PROGRAM Auto
VAR
	MovRightS: BOOL;
	MovRightL: BOOL;
	MovLeftS: BOOL;
	TON_Right: TON;
	TON_Left: TON;
	
	Home: BOOL;
	HomeMemory: BOOL;
	ManRequest: BOOL;
	TON_Right1: TON;
	TON_Left1: TON;
END_VAR
VAR // added by the converter: edge detectors and wires of the graphical bodies
    _w1 : BOOL;
END_VAR

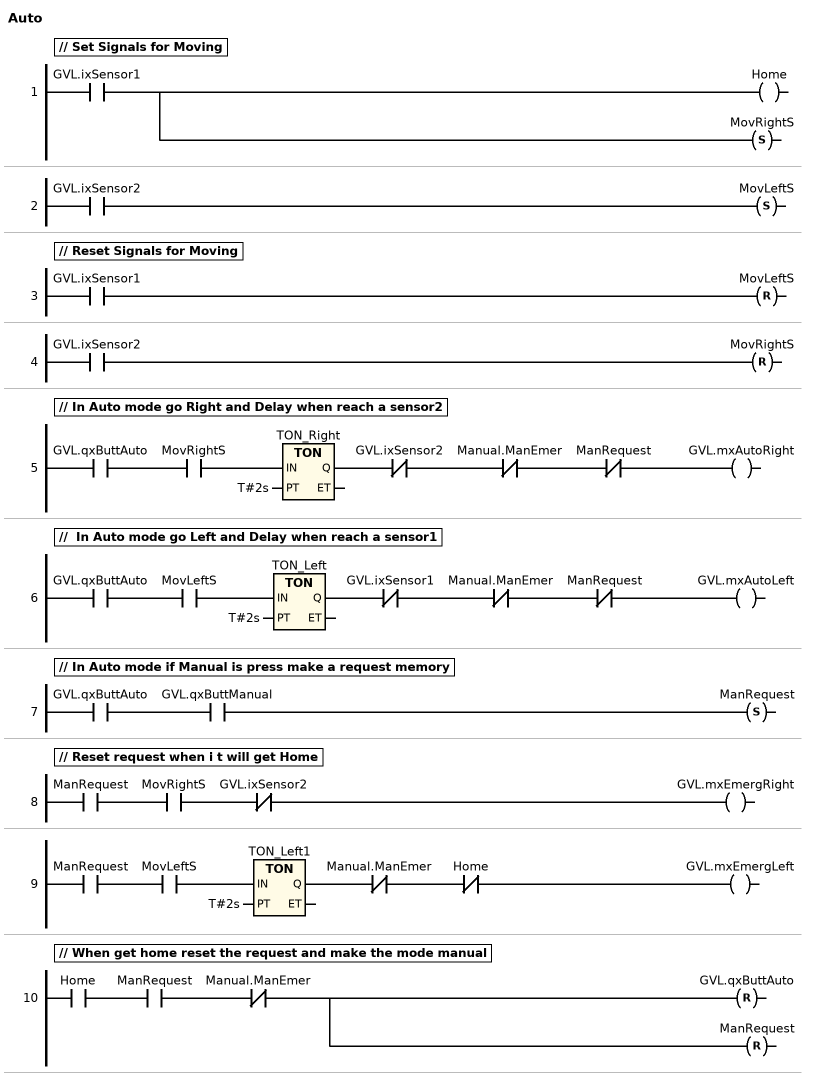
// NETWORK 1
// label: // Set Signals for Moving
Home := GVL.ixSensor1;
MovRightS S= GVL.ixSensor1;

// NETWORK 2
MovLeftS S= GVL.ixSensor2;

// NETWORK 3
// label: // Reset Signals for Moving
MovLeftS R= GVL.ixSensor1;

// NETWORK 4
MovRightS R= GVL.ixSensor2;

// NETWORK 5
// label: // In Auto mode go Right and Delay when reach a sensor2
TON_Right(IN := GVL.qxButtAuto AND MovRightS, PT := T#2s); // TON
GVL.mxAutoRight := TON_Right.Q AND NOT GVL.ixSensor2 AND NOT Manual.ManEmer AND NOT ManRequest;

// NETWORK 6
// label: //  In Auto mode go Left and Delay when reach a sensor1
TON_Left(IN := GVL.qxButtAuto AND MovLeftS, PT := T#2s); // TON
GVL.mxAutoLeft := TON_Left.Q AND NOT GVL.ixSensor1 AND NOT Manual.ManEmer AND NOT ManRequest;

// NETWORK 7
// label: // In Auto mode if Manual is press make a request memory
ManRequest S= GVL.qxButtAuto AND GVL.qxButtManual;

// NETWORK 8
// label: // Reset request when i t will get Home
GVL.mxEmergRight := ManRequest AND MovRightS AND NOT GVL.ixSensor2;

// NETWORK 9
TON_Left1(IN := ManRequest AND MovLeftS, PT := T#2s); // TON
GVL.mxEmergLeft := TON_Left1.Q AND NOT Manual.ManEmer AND NOT Home;

// NETWORK 10
// label: // When get home reset the request and make the mode manual
_w1 := Home AND ManRequest AND NOT Manual.ManEmer;
GVL.qxButtAuto R= _w1;
ManRequest R= _w1;

END_PROGRAM

(* stored: Version 1.1.0.1, ProductVersion 3.1.4024.12
   POU Auto: Id {07577967-2704-4b49-8a84-45396085dff0}, SpecialFunc None *)
